// TIA Portal V20 export
DATA_BLOCK "PM04"   // DB337
// stored: MemoryReserve 100
   VAR
      "STACK TABLE GAP PAD UP" : Bool := FALSE;
      "STACK TABLE GAP PAD DOWN" : Bool := FALSE;
      "CATHODE MANDREL CLAMP FRONT ON" : Bool := FALSE;
      SPARE : Bool := FALSE;
      "CATHODE MANDREL CLAMP REAR ON" : Bool := FALSE;
      SPARE_1 : Bool := FALSE;
      "ANODE MANDREL CLAMP FRONT ON" : Bool := FALSE;
      SPARE_2 : Bool := FALSE;
      "ANODE MANDREL CLAMP REAR ON" : Bool := FALSE;
   END_VAR
BEGIN
END_DATA_BLOCK
